Fanuc KAREL source: ko00039.KL

-- PROVISIONAL review KL for V770-1; original PC SHA256 f28c15513c74f95191319f0fefb32b4403e8db883475a56fe35e0e27faf65d23
-- Incomplete behavior may be omitted. Consult companion uncertainty JSON. Do not deploy.
PROGRAM KO00039
%NOLOCKGROUP
BEGIN
  -- UNRESOLVED_PC offsets 5-12; opcodes 9D,23
  -- UNRESOLVED_PC offsets 17-69; opcodes 27,27,49,7E,AD,27,49,7E,AD,22,31,7E,4A
  -- UNRESOLVED_PC offsets 74-78; opcodes 7F
END KO00039
